{attribute 'reflection'}
FUNCTION_BLOCK FB_BaseDevice IMPLEMENTS I_Device
VAR_INPUT
	safetyOK			: BOOL := TRUE;
END_VAR
VAR_OUTPUT
END_VAR
VAR
	{attribute 'instance-path'} 
    {attribute 'noinit'} 
    _sid				: STRING(255);
	_id					: WORD;
	_it					: I_Device;

	state				: INT;
	SM					: FB_StateManager;
	staleResetTm		: TON;
	staleResetTime		: TIME := T#1S;
	textState			: STRING(255) := 'Waiting for ready';

	msg					: FB_TcMessage;
END_VAR

///////////////////////////////////////////////////////////////////////////////
// FB_BaseDevice
//
// v1.0.0
//
// busy: Defaults to false
// done: Defaults to false
// error: Defaults to state < 0
// ready: Defaults to state >= 1000
///////////////////////////////////////////////////////////////////////////////

SM(state := state);
staleResetTm(IN := state <= -1000, PT := staleResetTime);

CASE state OF
	0:
		textState := 'Waiting for ready';
	999:
		textState := 'Idle';
	1000:
		textState := 'Running';
	-1:
		textState := 'Error';
	-1000:
		textState := 'Resetting';
END_CASE

METHOD PROTECTED FINAL alarm : BOOL
VAR_INPUT
	evt	: TcEventEntry;
END_VAR

alarm := alarmJson(evt, '');
END_METHOD

METHOD PROTECTED FINAL alarmAds : BOOL
VAR_INPUT
	errorId	: UDINT;
END_VAR

state := -1;
msg.Create(TC_EVENT_CLASSES.AdsEventClass, errorId, TcEventSeverity.Error, 0);
msg.Send(0);
END_METHOD

METHOD PROTECTED FINAL alarmJson : BOOL
VAR_INPUT
	evt	: TcEventEntry;
	str	: STRING(255);
END_VAR

state := -1;

msg.CreateEx(evt, 0);
IF len(str) > 0 THEN
	msg.SetJsonAttribute(str);
END_IF

msg.Send(0);
END_METHOD

{attribute 'monitoring' := 'variable'}
PROPERTY busy : BOOL
GET

busy := FALSE;
END_GET
END_PROPERTY

{attribute 'monitoring' := 'variable'}
PROPERTY done : BOOL
GET

done := FALSE;
END_GET
END_PROPERTY

{attribute 'monitoring' := 'variable'}
PROPERTY error : BOOL
GET

error := state < 0;
END_GET
END_PROPERTY

METHOD FB_init : BOOL
VAR_INPUT
	bInitRetains : BOOL; // if TRUE, the retain variables are initialized (warm start / cold start)
	bInCopyCode : BOOL;  // if TRUE, the instance afterwards gets moved into the copy code (online change)
END_VAR

_sid := F_RemoveProjectName(_sid);
_id := F_DATA_TO_CRC16_CCITT(ADR(_sid), TO_UDINT(len(_sid)), 0);
_it := THIS^;
{IF defined (variable: DH)}
DH.pushDevice(_sid, THIS);
{END_IF}

// Call release to help if the FB is made persistent
msg.Release();
END_METHOD

{attribute 'monitoring' := 'variable'}
PROPERTY id : DWORD
GET

id := _id;
END_GET
END_PROPERTY

METHOD PROTECTED FINAL message : BOOL
VAR_INPUT
	evt	: TcEventEntry;
END_VAR

message := messageJson(evt, '');
END_METHOD

METHOD PROTECTED FINAL messageJson : BOOL
VAR_INPUT
	evt	: TcEventEntry;
	str	: STRING(255);
END_VAR

msg.CreateEx(evt, 0);
IF len(str) > 0 THEN
	msg.SetJsonAttribute(str);
END_IF
msg.Send(0);
END_METHOD

{attribute 'monitoring' := 'variable'}
PROPERTY ready : BOOL
GET

ready := state >= 1000;
END_GET
END_PROPERTY

METHOD FINAL reset : BOOL
VAR_INPUT
END_VAR

IF state > -1000 OR staleResetTm.Q THEN
	staleResetTm(IN := FALSE);
	state := -1000;
END_IF
reset := ready;
END_METHOD

{attribute 'monitoring' := 'variable'}
PROPERTY FINAL sid : STRING(255)
GET

sid := _sid;
END_GET
END_PROPERTY

END_FUNCTION_BLOCK

(* stored: Version 1.1.0.1, ProductVersion 3.1.4024.10
   POU FB_BaseDevice: Id {be73e59d-4857-08fa-3e36-351227410420}, SpecialFunc None
   Method alarm: Id {547479bf-eb7a-0e41-38c3-d9036b80b96d}
   Method alarmAds: Id {12a1f46f-4bcc-418f-bbbe-02ec89e48c4a}
   Method alarmJson: Id {42163503-9fc5-4d79-bb03-d172f1f629b0}
   Property busy: Id {94db9ee7-d668-4770-be62-8756cd42f16a}
   Get Get: Id {35be04ff-0615-4caa-9b01-e949f67434d5}
   Property done: Id {2afd0192-49f4-4ef5-9a3c-93add18ec56f}
   Get Get: Id {0279e71b-27bb-4694-9cd9-444b6d88559d}
   Property error: Id {929ea1cf-9110-4108-98ea-1c70326ad33e}
   Get Get: Id {389bfdcc-eef7-4e60-8b5c-9617c918accc}
   Method FB_init: Id {99b621a9-3739-46f2-952f-366871f4a112}
   Property id: Id {3a772f72-99ed-4183-809c-1dd6935b6e56}
   Get Get: Id {f4a9844d-2d4c-455d-8cd7-58941e8e7b5f}
   Method message: Id {c856483f-6003-096c-24f5-5d5be41b8fd2}
   Method messageJson: Id {530a4aab-fe06-4a3c-94c5-00cf43921cfe}
   Property ready: Id {22fc3b10-1284-4368-bc38-fa18aa1d764b}
   Get Get: Id {c86111bc-91d2-456c-ae0f-6aa8da48b550}
   Method reset: Id {a592e39e-1d9b-0362-1d77-fe72b83d0b78}
   Property sid: Id {c5e28322-06de-4b54-bc30-afa6b52ad35f}
   Get Get: Id {3f8c8da3-5d07-48ab-9fe5-fd02f15544d8} *)
